FUNCTION_BLOCK ServoNC
VAR_INPUT CONSTANT
	bEnable : BOOL;
END_VAR
VAR_OUTPUT
	home AT %I* : BOOL;
	outerLimit AT %I* : BOOL;
	innerLimit AT %I* : BOOL;
	
	ready : BOOL;
	busy : BOOL;
	error : BOOL;
	homeSet : BOOL;
	
	position : LREAL;
END_VAR
VAR
	axis : AXIS_REF;
	
	mcReadPosition : MC_ReadActualPosition;
	mcReset : MC_Reset;
	
	mcPower : MC_Power;
	mcMoveAbsolute : MC_MoveAbsolute;
	mcMoveRelative : MC_MoveRelative;
	mcMoveVelocity : MC_MoveVelocity;
	
	mcStop : MC_Stop;
	mcSetPosition : MC_SetPosition;
	
	step : Homing;
END_VAR
VAR_STAT CONSTANT
	targetingVelocity : INT := 500;
	continuousVelocity : INT := 200;
END_VAR

mcReadPosition(
	Axis:= axis, 
	Enable:= TRUE, 
	Valid=> , 
	Busy=> , 
	Error=> , 
	ErrorID=> , 
	Position=> position);

mcReset(
	Axis:= axis, 
	Execute:= , 
	Done=> , 
	Busy=> , 
	Error=> , 
	ErrorID=> );

mcPower(
	Axis:= axis, 
	Enable:= bEnable, 
	Enable_Positive:= TRUE, 
	Enable_Negative:= TRUE, 
	Override:= 100, 
	BufferMode:= , 
	Options:= , 
	Status=> , 
	Busy=> , 
	Active=> , 
	Error=> , 
	ErrorID=> );

mcMoveAbsolute(
	Axis:= axis, 
	Execute:= , 
	Position:= , 
	Velocity:= targetingVelocity, 
	Acceleration:= , 
	Deceleration:= , 
	Jerk:= , 
	BufferMode:= , 
	Options:= , 
	Done=> , 
	Busy=> , 
	Active=> , 
	CommandAborted=> , 
	Error=> , 
	ErrorID=> );
		
mcMoveRelative(
	Axis:= axis, 
	Execute:= , 
	Distance:= ,
	Velocity:= targetingVelocity, 
	Acceleration:= , 
	Deceleration:= , 
	Jerk:= , 
	BufferMode:= , 
	Options:= , 
	Done=> , 
	Busy=> , 
	Active=> , 
	CommandAborted=> , 
	Error=> , 
	ErrorID=> );
	
mcMoveVelocity(
	Axis:= axis, 
	Execute:= , 
	Velocity:= continuousVelocity, 
	Acceleration:= , 
	Deceleration:= , 
	Jerk:= , 
	Direction:= , 
	BufferMode:= , 
	Options:= , 
	InVelocity=> , 
	Busy=> , 
	Active=> , 
	CommandAborted=> , 
	Error=> , 
	ErrorID=> );
	
mcStop(
	Axis:= axis, 
	Execute:= , 
	Deceleration:= , 
	Jerk:= , 
	Options:= , 
	Done=> , 
	Busy=> , 
	Active=> , 
	CommandAborted=> , 
	Error=> , 
	ErrorID=> );

mcSetPosition(
	Axis:= axis, 
	Execute:= , 
	Position:= , 
	Mode:= , 
	Options:= , 
	Done=> , 
	Busy=> , 
	Error=> , 
	ErrorID=> );
	
busy := mcMoveAbsolute.Busy OR mcMoveRelative.Busy OR mcMoveVelocity.Busy OR mcSetPosition.Busy OR mcReset.Busy OR mcStop.Busy OR step <> 0;
error := mcMoveAbsolute.Error OR mcMoveRelative.Error OR mcMoveVelocity.Error OR mcSetPosition.Error OR mcReset.Error OR mcStop.Error OR step <> 0;
ready := bEnable AND NOT busy AND homeSet;

IF step <> 0 THEN
	mcReset.Execute := FALSE;
	mcMoveAbsolute.Execute := FALSE;
	mcMoveRelative.Execute := FALSE;
	mcMoveVelocity.Execute := FALSE;
	mcStop.Execute := FALSE;
	mcSetPosition.Execute := FALSE;
END_IF

METHOD homingSequence : BOOL
CASE step OF
	Homing.IDLE:
		IF bEnable THEN
			step := Homing.REDO;
		END_IF
		
	Homing.REDO:
		IF mcMoveVelocity.Execute AND NOT innerLimit THEN
			mcMoveVelocity.Execute := FALSE;
			step := Homing.HOME_OUT;
			RETURN;
		END_IF
		
		mcMoveVelocity.Direction := MC_Negative_Direction;
		mcMoveVelocity.Execute := TRUE;
		
	Homing.HOME_OUT:
		IF mcMoveVelocity.Execute AND NOT home THEN //if reached home
			mcMoveVelocity.Execute := FALSE;
			step := Homing.STOP;
			RETURN;
		END_IF
		
		mcMoveVelocity.Direction := MC_Positive_Direction;
		mcMoveVelocity.Execute := TRUE;
		
	Homing.STOP:
		IF mcStop.Execute AND mcStop.Done THEN
			mcStop.Execute := FALSE;
			step := Homing.SET;
			RETURN;
		END_IF
		
		mcStop.Execute := TRUE;
		
	Homing.SET:
		IF mcSetPosition.Execute AND mcSetPosition.Done THEN
			mcSetPosition.Execute := FALSE;
			homingSequence := TRUE;
			step := Homing.IDLE;
			RETURN;
		END_IF
		
		mcSetPosition.Position := 0;
		mcSetPosition.Execute := TRUE;
		
END_CASE
END_METHOD

METHOD moveAbsolute : BOOL
VAR_INPUT
	targetPos : LREAL;
END_VAR
IF NOT busy AND NOT error THEN
	mcMoveAbsolute.Position := targetPos;
END_IF
moveAbsolute := mcMoveAbsolute.Done;
END_METHOD

METHOD moveContinuous : BOOL
VAR_INPUT
	direction : MC_Direction;
END_VAR
mcMoveVelocity.Direction := direction;

mcMoveVelocity.Execute := TRUE;

moveContinuous := NOT mcMoveVelocity.Error;
END_METHOD

METHOD moveRelative : BOOL
VAR_INPUT
	distance : LREAL;
END_VAR
mcMoveRelative.Distance := distance;

moveRelative := mcMoveRelative.Done;
END_METHOD

METHOD reset : BOOL
VAR_INPUT
END_VAR
mcReset.Execute := TRUE;

reset := mcReset.Done;
END_METHOD

METHOD stop : BOOL
VAR_INPUT
END_VAR
END_METHOD

END_FUNCTION_BLOCK

(* stored: Version 1.1.0.1, ProductVersion 3.1.4024.11
   POU ServoNC: Id {f939ae28-30bd-4997-8b95-af50702e8d64}, SpecialFunc None
   Method homingSequence: Id {c889c79b-08e7-46ba-b03a-e3652fe9a7a9}
   Method moveAbsolute: Id {9a0c1523-e496-48d2-89d9-d71629c86307}
   Method moveContinuous: Id {c1bd97e2-f7e7-45ed-bf81-7afd3b7c53ff}
   Method moveRelative: Id {a4516e41-c115-4d38-aa54-f9462db8dc0d}
   Method reset: Id {b7706fbc-8e49-4562-bc6d-21f87f45b14e}
   Method stop: Id {131a01d5-9f85-446c-9242-ad02c99596c6} *)
